VAR_GLOBAL CONSTANT
    MAX_TESTS : DINT := 200;
END_VAR

(* stored: Version 1.1.0.1, ProductVersion 3.1.4024.11
   GVL Parameters: Id {5ac96168-fae9-4200-ac5c-82709ff5d76a}, ParameterList True *)
